(*
  QualiVision line camera system
  DMAX106.   
*)
FUNCTION_BLOCK FB_LineCamera106 EXTENDS FB_LineCamera

VAR CONSTANT
  cCameraWidth106           : DINT := 13440;   (*Camera width [px]*)
  cCameraMechOffsetTC106    : REAL :=  88.0;   (*Camera mechanical offset at calibration temp [mm]*)
  cMechOffsetCameraToPU106  : REAL :=  30.31;  (*Camera mechanical offset to PrintUnit [mm]*)
  cPrintUnitMechOffsetTC106 : REAL := 31.4747; (*PrintUnit mechanical offset at calibration temp [mm]*)
END_VAR

SUPER^();

METHOD InitLineCamera
VAR_INPUT
  nPrintUnitResolution         : UDINT;    (*printhead pixel resolution [dpi]*)
  nPrintUnitSubPx              : UDINT;    (*print unit subPixel resolution [SubPx]*)
  nPrintUnitWidth              : UDINT;    (*print unit width in [px]*)
  iCameraTrigger               : I_CameraTrigger;
END_VAR
(*Init for dmax type*)
_nCameraWidth           := cCameraWidth106;
_fCameraMechOffsetTC    := cCameraMechOffsetTC106;
_fMechOffsetCameraToPU  := cMechOffsetCameraToPU106;
_fPrintUnitMechOffsetTC := cPrintUnitMechOffsetTC106;

SUPER^.InitLineCamera( nPrintUnitResolution := nPrintUnitResolution
                      , nPrintUnitSubPx := nPrintUnitSubPx
                      , nPrintUnitWidth := nPrintUnitWidth
                      , iCameraTrigger := iCameraTrigger);
END_METHOD

{attribute 'monitoring':='variable'}
PROPERTY sName : STRING
GET
sName := 'LineCam 106';
END_GET
END_PROPERTY

END_FUNCTION_BLOCK

(* stored: Version 1.1.0.1, ProductVersion 3.1.4024.3
   POU FB_LineCamera106: Id {eed955d2-a1f9-4a17-b849-a639a208bf07}, SpecialFunc None
   Method InitLineCamera: Id {695e7c1d-784c-491a-a112-3e3dd542606f}
   Property sName: Id {4c93f93f-64fc-4113-a181-8344eee37c29}
   Get Get: Id {0267b6a1-d2d5-4f89-899f-b45bf1112108} *)
